FUNCTION_BLOCK PhaseObjTest (* CAT Function Block Type *)
  (* Standard: 61499-2 *)
  (* Version 0.0, 6/5/2026, Schneider Electric, template *)
  PACKAGE SE.Nereda;
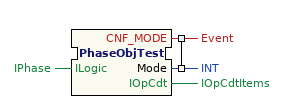
  EVENT_OUTPUT
    CNF_MODE WITH Mode;
  END_EVENT
  VAR_OUTPUT
    Mode : INT;
  END_VAR
  SOCKETS
    ILogic : IPhase;
  END_SOCKETS
  PLUGS
    IOpCdt : IOpCdtItems;
  END_PLUGS
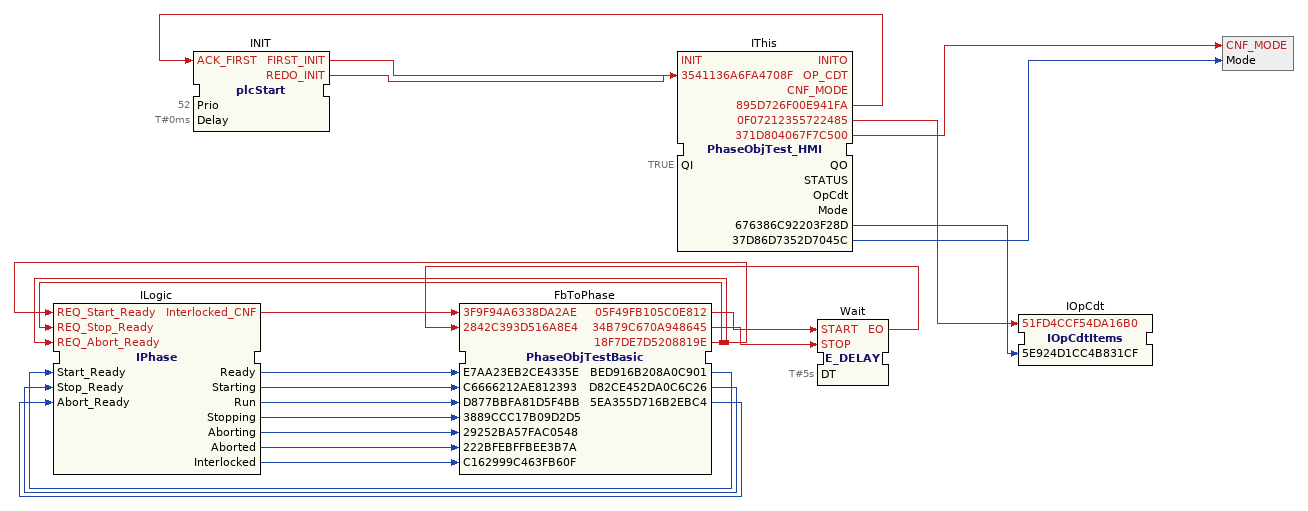
  FBS
    IThis : PhaseObjTest_HMI(QI := TRUE);
    FbToPhase : PhaseObjTestBasic;
    Wait : E_DELAY(DT := T#5s);
    INIT : plcStart(Prio := 52, Delay := T#0ms);
  END_FBS
  EVENT_CONNECTIONS
    ILogic.Interlocked_CNF TO FbToPhase.3F9F94A6338DA2AE;
    FbToPhase.05F49FB105C0E812 TO Wait.START;
    FbToPhase.34B79C670A948645 TO Wait.STOP;
    Wait.EO TO FbToPhase.2842C393D516A8E4;
    FbToPhase.18F7DE7D5208819E TO ILogic.REQ_Start_Ready;
    FbToPhase.18F7DE7D5208819E TO ILogic.REQ_Stop_Ready;
    FbToPhase.18F7DE7D5208819E TO ILogic.REQ_Abort_Ready;
    INIT.FIRST_INIT TO IThis.3541136A6FA4708F;
    INIT.REDO_INIT TO IThis.3541136A6FA4708F;
    IThis.895D726F00E941FA TO INIT.ACK_FIRST;
    IThis.0F07212355722485 TO IOpCdt.51FD4CCF54DA16B0;
    IThis.371D804067F7C500 TO CNF_MODE;
  END_CONNECTIONS
  DATA_CONNECTIONS
    ILogic.Ready TO FbToPhase.E7AA23EB2CE4335E;
    ILogic.Starting TO FbToPhase.C6666212AE812393;
    ILogic.Run TO FbToPhase.D877BBFA81D5F4BB;
    ILogic.Stopping TO FbToPhase.3889CCC17B09D2D5;
    ILogic.Aborting TO FbToPhase.29252BA57FAC0548;
    ILogic.Aborted TO FbToPhase.222BFEBFFBEE3B7A;
    ILogic.Interlocked TO FbToPhase.C162999C463FB60F;
    FbToPhase.BED916B208A0C901 TO ILogic.Start_Ready;
    FbToPhase.D82CE452DA0C6C26 TO ILogic.Stop_Ready;
    FbToPhase.5EA355D716B2EBC4 TO ILogic.Abort_Ready;
    IThis.676386C92203F28D TO IOpCdt.5E924D1CC4B831CF;
    IThis.37D86D7352D7045C TO Mode;
  END_CONNECTIONS
END_FUNCTION_BLOCK
